// TIA Portal project "babu_4WayTrafficIndian" (V15)

(* hardware
DEVICE "S7-1200 station_1"  S7-1200 Station
   slot 0: "Rack_0"  S7-1200 Rack  Rack  V1.0
   slot 1: "PLC_1"  CPU 1212C DC/DC/DC  6ES7 212-1AE40-0XB0  V4.2
*)

// ===== PLC "PLC_1"  CPU 1212C DC/DC/DC =====

VAR_GLOBAL   // PLC tag table "Default tag table"
   "POWER BUTTON" AT %I0.0 : Bool;
   "POWER BUTTON MEMORY" AT %M0.1 : Bool;
   "INITIALIZE" AT %M0.2 : Bool;
   "IP2" AT %M0.3 : Bool;
   "OP2" AT %Q0.0 : Bool;
   "IP21" AT %M0.4 : Bool;
   "PP MEMORY" AT %M0.5 : Bool;
   "G3M" AT %M0.6 : Bool;
   "G1M" AT %M0.7 : Bool;
   "G2M" AT %M1.0 : Bool;
   "Y1M" AT %M1.1 : Bool;
   "Y2M" AT %M1.2 : Bool;
   "Y3M" AT %M1.3 : Bool;
   "R1M" AT %M1.4 : Bool;
   "R2M" AT %M1.5 : Bool;
   "R3M" AT %M1.6 : Bool;
   "G1" AT %Q0.1 : Bool;
   "G2" AT %Q0.2 : Bool;
   "G3" AT %Q0.3 : Bool;
   "Y1" AT %Q0.4 : Bool;
   "Y2" AT %Q0.5 : Bool;
   "Y3" AT %Q0.6 : Bool;
   "R1" AT %Q0.7 : Bool;
   "R2" AT %Q1.0 : Bool;
   "R3" AT %Q1.1 : Bool;
   "SEQ1" AT %M0.0 : Bool;
   "SEQ2" AT %M1.7 : Bool;
   "SEQ3" AT %M2.0 : Bool;
   "SEQ4" AT %M2.1 : Bool;
   "SEQ5" AT %M2.2 : Bool;
   "SEQ6" AT %M2.3 : Bool;
   "ERROR" AT %M2.4 : Bool;
   "IP22" AT %M2.5 : Bool;
   "IP22MEM" AT %M2.6 : Bool;
   "OP22" AT %M2.7 : Bool;
   "IP23" AT %M3.0 : Bool;
   "IP24" AT %M3.1 : Bool;
   "IP24MEM" AT %M3.2 : Bool;
   "OP24" AT %Q1.2 : Bool;
   "PP MEM 1" AT %M3.3 : Bool;
   "PP MEM 2" AT %M3.4 : Bool;
   "PP MEM 3" AT %M3.5 : Bool;
   "PP MEM 4" AT %M3.6 : Bool;
   "PP MEM5" AT %M3.7 : Bool;
   "PP MEM6" AT %M4.0 : Bool;
   "PP MEM7" AT %M4.1 : Bool;
   "PP MEM8" AT %M4.2 : Bool;
   "PP MEM9" AT %M4.3 : Bool;
   "SEQ7" AT %M4.4 : Bool;
   "SEQ8" AT %M4.5 : Bool;
   "SEQ9" AT %M4.6 : Bool;
   "R4M" AT %M4.7 : Bool;
   "G4M" AT %M5.0 : Bool;
   "Y4M" AT %M5.1 : Bool;
   "R4" AT %Q5.2 : Bool;
   "G4" AT %Q5.3 : Bool;
   "Y4" AT %Q5.4 : Bool;
END_VAR

// folder: System blocks/Program resources

DATA_BLOCK "IEC_Timer_0_DB"   // DB1
{ S7_Optimized_Access := 'TRUE' }
AUTHOR : Simatic
FAMILY : IEC
NAME : IEC_TMR
VERSION : 1.0
// stored: InstanceOfName IEC_TIMER
"IEC_TIMER"
BEGIN
END_DATA_BLOCK

DATA_BLOCK "IEC_Timer_0_DB_2"   // DB3
{ S7_Optimized_Access := 'TRUE' }
AUTHOR : Simatic
FAMILY : IEC
NAME : IEC_TMR
VERSION : 1.0
// stored: InstanceOfName IEC_TIMER
"IEC_TIMER"
BEGIN
END_DATA_BLOCK

DATA_BLOCK "IEC_Timer_0_DB_3"   // DB4
{ S7_Optimized_Access := 'TRUE' }
AUTHOR : Simatic
FAMILY : IEC
NAME : IEC_TMR
VERSION : 1.0
// stored: InstanceOfName IEC_TIMER
"IEC_TIMER"
BEGIN
END_DATA_BLOCK

DATA_BLOCK "IEC_Timer_0_DB_4"   // DB5
{ S7_Optimized_Access := 'TRUE' }
AUTHOR : Simatic
FAMILY : IEC
NAME : IEC_TMR
VERSION : 1.0
// stored: InstanceOfName IEC_TIMER
"IEC_TIMER"
BEGIN
END_DATA_BLOCK

DATA_BLOCK "IEC_Timer_0_DB_5"   // DB6
{ S7_Optimized_Access := 'TRUE' }
AUTHOR : Simatic
FAMILY : IEC
NAME : IEC_TMR
VERSION : 1.0
// stored: InstanceOfName IEC_TIMER
"IEC_TIMER"
BEGIN
END_DATA_BLOCK

DATA_BLOCK "IEC_Timer_0_DB_7"   // DB8
{ S7_Optimized_Access := 'TRUE' }
AUTHOR : Simatic
FAMILY : IEC
NAME : IEC_TMR
VERSION : 1.0
// stored: InstanceOfName IEC_TIMER
"IEC_TIMER"
BEGIN
END_DATA_BLOCK

// folder: (top level)

ORGANIZATION_BLOCK "Main"   // OB1, LAD, ProgramCycle
TITLE = "Main Program Sweep (Cycle)"
{ S7_Optimized_Access := 'TRUE' }
VERSION : 0.1
   VAR_INPUT
      Initial_Call : Bool;   // Initial call of this OB
      Remanence : Bool;   // =True, if remanent data are available
   END_VAR
   VAR_TEMP   // added for the SCL form of the ladder/FBD networks
      _w1 : Bool;
      _w2 : Bool;
      _w3 : Bool;
   END_VAR
BEGIN

REGION Network 1: POWER UP
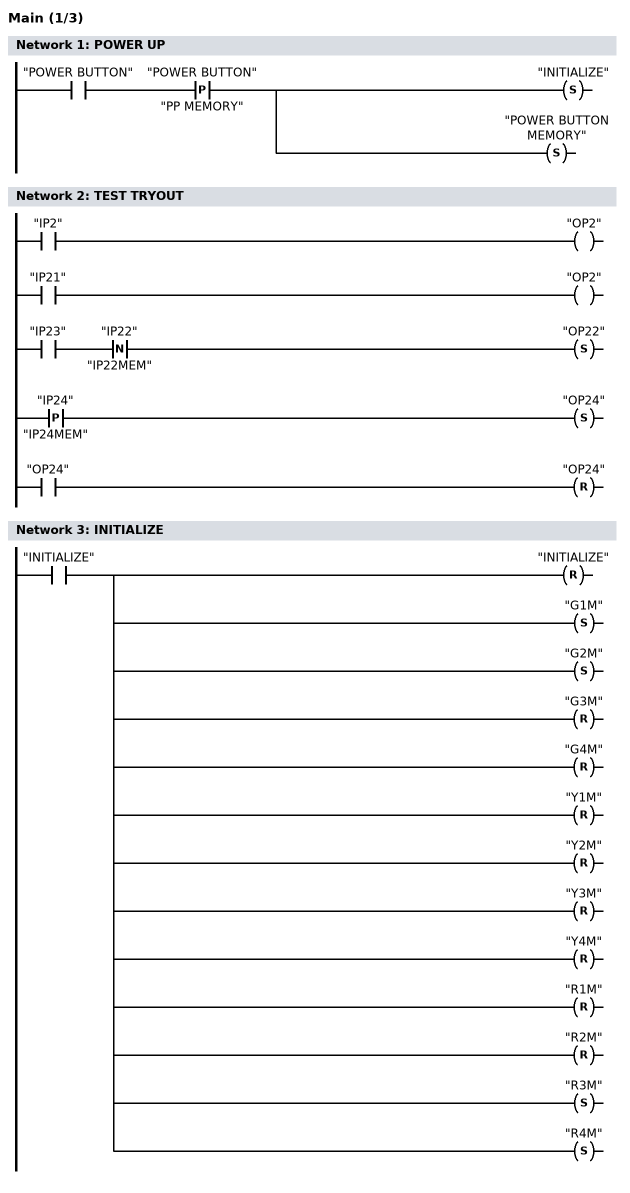
   RUNG wire#powerrail
      Contact( "POWER BUTTON" )
      P_Contact(operand := "POWER BUTTON", bit := "PP MEMORY")
      wire#w1
      S_Coil( "INITIALIZE" )
   END_RUNG
   RUNG wire#w1
      S_Coil( "POWER BUTTON MEMORY" )
   END_RUNG
   // the same network as SCL:
   #_w1 := "POWER BUTTON" AND "POWER BUTTON" AND NOT "PP MEMORY";   // rising edge of "POWER BUTTON"
   "PP MEMORY" := "POWER BUTTON";
   IF #_w1 THEN
       "INITIALIZE" := TRUE;
       "POWER BUTTON MEMORY" := TRUE;
   END_IF;
END_REGION

REGION Network 2: TEST TRYOUT
   RUNG wire#powerrail
      Contact( "IP2" )
      Coil( "OP2" )
   END_RUNG
   RUNG wire#powerrail
      Contact( "IP21" )
      Coil( "OP2" )
   END_RUNG
   RUNG wire#powerrail
      Contact( "IP23" )
      N_Contact(operand := "IP22", bit := "IP22MEM")
      S_Coil( "OP22" )
   END_RUNG
   RUNG wire#powerrail
      P_Contact(operand := "IP24", bit := "IP24MEM")
      S_Coil( "OP24" )
   END_RUNG
   RUNG wire#powerrail
      Contact( "OP24" )
      R_Coil( "OP24" )
   END_RUNG
   // the same network as SCL:
   "OP2" := "IP2";
   "OP2" := "IP21";
   #_w1 := "IP23" AND NOT "IP22" AND "IP22MEM";   // falling edge of "IP22"
   "IP22MEM" := "IP22";
   IF #_w1 THEN "OP22" := TRUE; END_IF;
   #_w2 := "IP24" AND NOT "IP24MEM";   // rising edge of "IP24"
   "IP24MEM" := "IP24";
   IF #_w2 THEN "OP24" := TRUE; END_IF;
   IF "OP24" THEN "OP24" := FALSE; END_IF;
END_REGION

REGION Network 3: INITIALIZE
   RUNG wire#powerrail
      Contact( "INITIALIZE" )
      wire#w1
      R_Coil( "INITIALIZE" )
   END_RUNG
   RUNG wire#w1
      S_Coil( "G1M" )
   END_RUNG
   RUNG wire#w1
      S_Coil( "G2M" )
   END_RUNG
   RUNG wire#w1
      R_Coil( "G3M" )
   END_RUNG
   RUNG wire#w1
      R_Coil( "G4M" )
   END_RUNG
   RUNG wire#w1
      R_Coil( "Y1M" )
   END_RUNG
   RUNG wire#w1
      R_Coil( "Y2M" )
   END_RUNG
   RUNG wire#w1
      R_Coil( "Y3M" )
   END_RUNG
   RUNG wire#w1
      R_Coil( "Y4M" )
   END_RUNG
   RUNG wire#w1
      R_Coil( "R1M" )
   END_RUNG
   RUNG wire#w1
      R_Coil( "R2M" )
   END_RUNG
   RUNG wire#w1
      S_Coil( "R3M" )
   END_RUNG
   RUNG wire#w1
      S_Coil( "R4M" )
   END_RUNG
   // the same network as SCL:
   #_w1 := "INITIALIZE";
   IF #_w1 THEN
       "INITIALIZE" := FALSE;
       "G1M" := TRUE;
       "G2M" := TRUE;
       "G3M" := FALSE;
       "G4M" := FALSE;
       "Y1M" := FALSE;
       "Y2M" := FALSE;
       "Y3M" := FALSE;
       "Y4M" := FALSE;
       "R1M" := FALSE;
       "R2M" := FALSE;
       "R3M" := TRUE;
       "R4M" := TRUE;
   END_IF;
END_REGION

REGION Network 4: OUTPUT
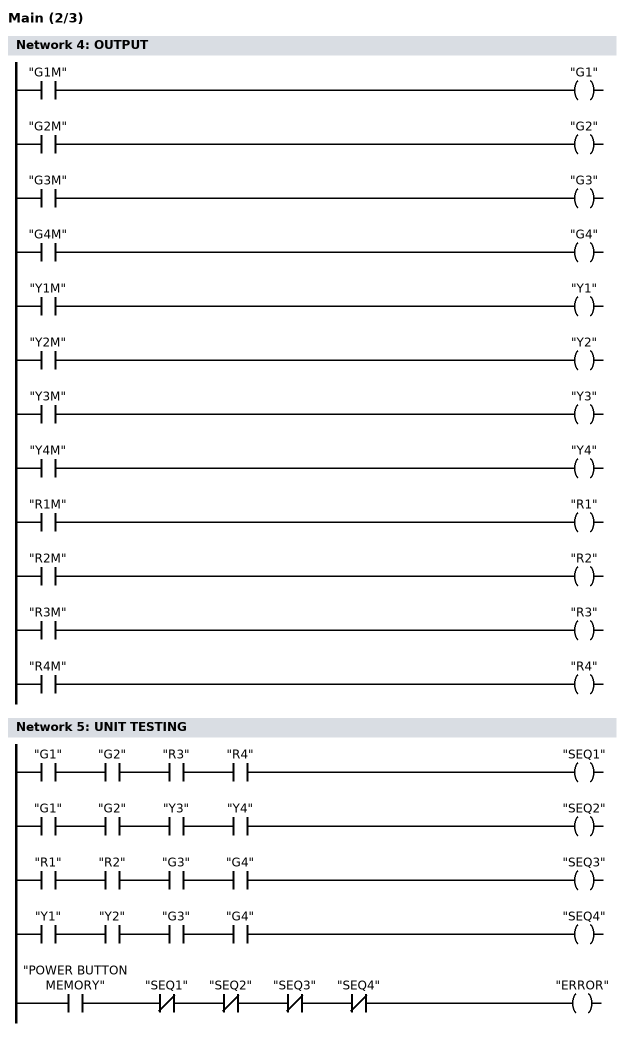
   RUNG wire#powerrail
      Contact( "G1M" )
      Coil( "G1" )
   END_RUNG
   RUNG wire#powerrail
      Contact( "G2M" )
      Coil( "G2" )
   END_RUNG
   RUNG wire#powerrail
      Contact( "G3M" )
      Coil( "G3" )
   END_RUNG
   RUNG wire#powerrail
      Contact( "G4M" )
      Coil( "G4" )
   END_RUNG
   RUNG wire#powerrail
      Contact( "Y1M" )
      Coil( "Y1" )
   END_RUNG
   RUNG wire#powerrail
      Contact( "Y2M" )
      Coil( "Y2" )
   END_RUNG
   RUNG wire#powerrail
      Contact( "Y3M" )
      Coil( "Y3" )
   END_RUNG
   RUNG wire#powerrail
      Contact( "Y4M" )
      Coil( "Y4" )
   END_RUNG
   RUNG wire#powerrail
      Contact( "R1M" )
      Coil( "R1" )
   END_RUNG
   RUNG wire#powerrail
      Contact( "R2M" )
      Coil( "R2" )
   END_RUNG
   RUNG wire#powerrail
      Contact( "R3M" )
      Coil( "R3" )
   END_RUNG
   RUNG wire#powerrail
      Contact( "R4M" )
      Coil( "R4" )
   END_RUNG
   // the same network as SCL:
   "G1" := "G1M";
   "G2" := "G2M";
   "G3" := "G3M";
   "G4" := "G4M";
   "Y1" := "Y1M";
   "Y2" := "Y2M";
   "Y3" := "Y3M";
   "Y4" := "Y4M";
   "R1" := "R1M";
   "R2" := "R2M";
   "R3" := "R3M";
   "R4" := "R4M";
END_REGION

REGION Network 5: UNIT TESTING
   RUNG wire#powerrail
      Contact( "G1" )
      Contact( "G2" )
      Contact( "R3" )
      Contact( "R4" )
      Coil( "SEQ1" )
   END_RUNG
   RUNG wire#powerrail
      Contact( "G1" )
      Contact( "G2" )
      Contact( "Y3" )
      Contact( "Y4" )
      Coil( "SEQ2" )
   END_RUNG
   RUNG wire#powerrail
      Contact( "R1" )
      Contact( "R2" )
      Contact( "G3" )
      Contact( "G4" )
      Coil( "SEQ3" )
   END_RUNG
   RUNG wire#powerrail
      Contact( "Y1" )
      Contact( "Y2" )
      Contact( "G3" )
      Contact( "G4" )
      Coil( "SEQ4" )
   END_RUNG
   RUNG wire#powerrail
      Contact( "POWER BUTTON MEMORY" )
      I_Contact( "SEQ1" )
      I_Contact( "SEQ2" )
      I_Contact( "SEQ3" )
      I_Contact( "SEQ4" )
      Coil( "ERROR" )
   END_RUNG
   // the same network as SCL:
   "SEQ1" := "G1" AND "G2" AND "R3" AND "R4";
   "SEQ2" := "G1" AND "G2" AND "Y3" AND "Y4";
   "SEQ3" := "R1" AND "R2" AND "G3" AND "G4";
   "SEQ4" := "Y1" AND "Y2" AND "G3" AND "G4";
   "ERROR" := "POWER BUTTON MEMORY" AND NOT "SEQ1" AND NOT "SEQ2" AND NOT "SEQ3" AND NOT "SEQ4";
END_REGION

REGION Network 6: G1 G2
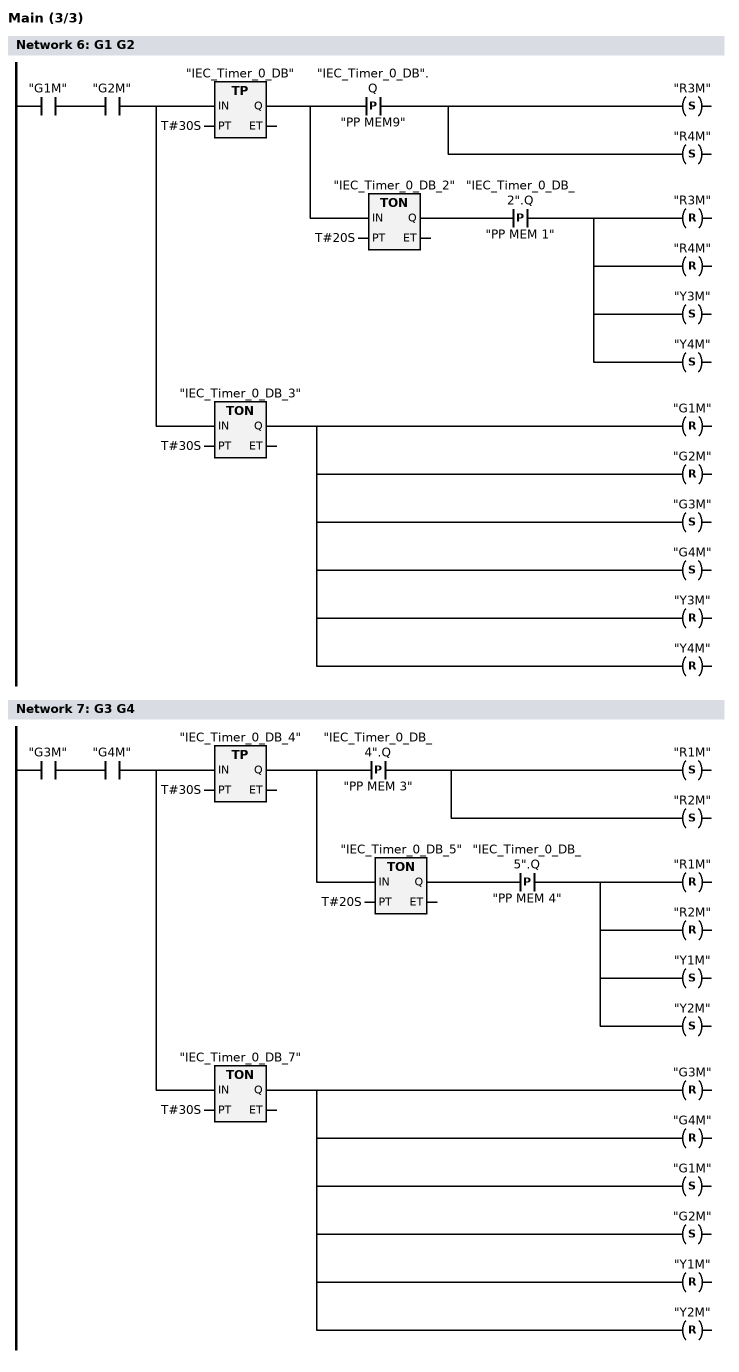
   #_w1 := "G1M" AND "G2M";
   "IEC_Timer_0_DB".TP(IN := #_w1, PT := T#30S);
   #_w2 := "IEC_Timer_0_DB".Q AND "IEC_Timer_0_DB".Q AND NOT "PP MEM9";   // rising edge of "IEC_Timer_0_DB".Q
   "PP MEM9" := "IEC_Timer_0_DB".Q;
   IF #_w2 THEN
       "R3M" := TRUE;
       "R4M" := TRUE;
   END_IF;
   "IEC_Timer_0_DB_2".TON(IN := "IEC_Timer_0_DB".Q, PT := T#20S);
   #_w3 := "IEC_Timer_0_DB_2".Q AND "IEC_Timer_0_DB_2".Q AND NOT "PP MEM 1";   // rising edge of "IEC_Timer_0_DB_2".Q
   "PP MEM 1" := "IEC_Timer_0_DB_2".Q;
   IF #_w3 THEN
       "R3M" := FALSE;
       "R4M" := FALSE;
       "Y3M" := TRUE;
       "Y4M" := TRUE;
   END_IF;
   "IEC_Timer_0_DB_3".TON(IN := #_w1, PT := T#30S);
   IF "IEC_Timer_0_DB_3".Q THEN
       "G1M" := FALSE;
       "G2M" := FALSE;
       "G3M" := TRUE;
       "G4M" := TRUE;
       "Y3M" := FALSE;
       "Y4M" := FALSE;
   END_IF;
END_REGION

REGION Network 7: G3 G4
   #_w1 := "G3M" AND "G4M";
   "IEC_Timer_0_DB_4".TP(IN := #_w1, PT := T#30S);
   #_w2 := "IEC_Timer_0_DB_4".Q AND "IEC_Timer_0_DB_4".Q AND NOT "PP MEM 3";   // rising edge of "IEC_Timer_0_DB_4".Q
   "PP MEM 3" := "IEC_Timer_0_DB_4".Q;
   IF #_w2 THEN
       "R1M" := TRUE;
       "R2M" := TRUE;
   END_IF;
   "IEC_Timer_0_DB_5".TON(IN := "IEC_Timer_0_DB_4".Q, PT := T#20S);
   #_w3 := "IEC_Timer_0_DB_5".Q AND "IEC_Timer_0_DB_5".Q AND NOT "PP MEM 4";   // rising edge of "IEC_Timer_0_DB_5".Q
   "PP MEM 4" := "IEC_Timer_0_DB_5".Q;
   IF #_w3 THEN
       "R1M" := FALSE;
       "R2M" := FALSE;
       "Y1M" := TRUE;
       "Y2M" := TRUE;
   END_IF;
   "IEC_Timer_0_DB_7".TON(IN := #_w1, PT := T#30S);
   IF "IEC_Timer_0_DB_7".Q THEN
       "G3M" := FALSE;
       "G4M" := FALSE;
       "G1M" := TRUE;
       "G2M" := TRUE;
       "Y1M" := FALSE;
       "Y2M" := FALSE;
   END_IF;
END_REGION
END_ORGANIZATION_BLOCK